// SIMATIC S7-200 SMART project (STEP 7-Micro/WIN SMART), CPU ST40

ORGANIZATION_BLOCK MAIN:OB1
TITLE=Program Comments
BEGIN
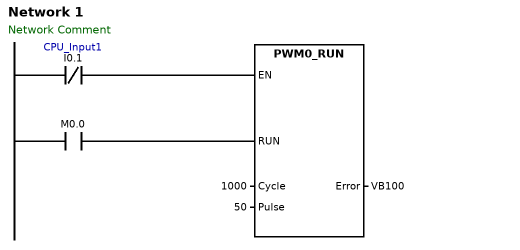
Network 1
// Network Comment
LDN    CPU_Input1:I0.1
=      L60.0
LD     M0.0
=      L63.7
LD     L60.0
CALL   PWM0_RUN:SBR1, L63.7, 1000, 50, VB100
END_ORGANIZATION_BLOCK

SUBROUTINE_BLOCK SBR_0:SBR0
TITLE=Subroutine Comments
BEGIN
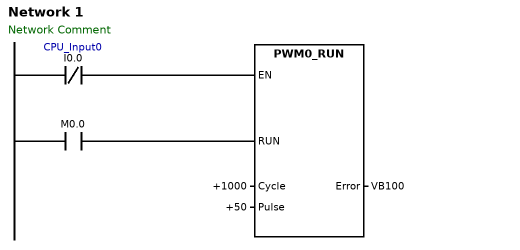
Network 1
// Network Comment
LDN    CPU_Input0:I0.0
=      L60.0
LD     M0.0
=      L63.7
LD     L60.0
CALL   PWM0_RUN:SBR1, L63.7, +1000, +50, VB100
END_SUBROUTINE_BLOCK

// SBR1: protected block, not included
